// TIA Portal V20 export
DATA_BLOCK "BK20"   // DB267
// stored: MemoryReserve 100
   VAR
      "X10-1 INS TRANSFER P&P1 X-AXIS LIMIT SENSOR(-)" : Bool;
      "X11-1 INS TRANSFER P&P1 X-AXIS LIMIT SENSOR(+)" : Bool;
      "X12-1 INS TRANSFER P&P2 X-AXIS LIMIT SENSOR(-)" : Bool;
      "X13-1 INS TRANSFER P&P2 X-AXIS LIMIT SENSOR(+)" : Bool;
      "X14-1 SPARE" : Bool;
      "X15-1 SPARE" : Bool;
      "X16-1 SPARE" : Bool;
      "X17-1 SPARE" : Bool;
      "X10-2 INS TRANSFER P&P1 X-AXIS HOMING SENSOR" : Bool;
      "X11-2 SPARE" : Bool;
      "X12-2 INS TRANSFER P&P2 X-AXIS HOMING SENSOR" : Bool;
      "X13-2 SPARE" : Bool;
      "X14-2 SPARE" : Bool;
      "X15-2 SPARE" : Bool;
      "X16-2 SPARE" : Bool;
      "X17-2 SPARE" : Bool;
   END_VAR
BEGIN
END_DATA_BLOCK
